FUNCTION_BLOCK AlarmNotAck (* Basic Function Block Type *)
  (* Standard: 61499-2 *)
  (* Version 0.0, 8/5/2026, Schneider Electric, Template *)
  PACKAGE SE.Nereda;
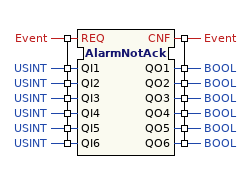
  EVENT_INPUT
    REQ WITH QI1, QI2, QI3, QI4, QI5, QI6; (* Normal Execution Request *)
  END_EVENT
  EVENT_OUTPUT
    CNF WITH QO1, QO2, QO3, QO4, QO5, QO6; (* Execution Confirmation *)
  END_EVENT
  VAR_INPUT
    QI1 : USINT; (* Input event qualifier *)
    QI2 : USINT;
    QI3 : USINT;
    QI4 : USINT;
    QI5 : USINT;
    QI6 : USINT;
  END_VAR
  VAR_OUTPUT
    QO1 : BOOL; (* Output event qualifier *)
    QO2 : BOOL;
    QO3 : BOOL;
    QO4 : BOOL;
    QO5 : BOOL;
    QO6 : BOOL;
  END_VAR
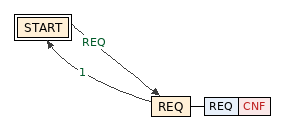
  EC_STATES
    START; (* Initial State *)
    REQ : REQ -> CNF; (* Normal execution *)
  END_STATES
  EC_TRANSITIONS
    START TO REQ := REQ;
    REQ TO START := 1;
  END_TRANSITIONS
  ALGORITHM INIT IN ST: (* Initialization algorithm *)
;
  END_ALGORITHM
  ALGORITHM REQ IN ST: (* Normally executed algorithm *)
;
IF QI1 = 2 THEN
	QO1 := TRUE;
ELSIF QI1 = 0 THEN
	QO1 := FALSE;
END_IF;

IF QI2 = 2 THEN
	QO2 := TRUE;
ELSIF QI2 = 0 THEN
	QO2 := FALSE;
END_IF;

IF QI3 = 2 THEN
	QO3 := TRUE;
ELSIF QI3 = 0 THEN
	QO3 := FALSE;
END_IF;

IF QI4 = 2 THEN
	QO4 := TRUE;
ELSIF QI4 = 0 THEN
	QO4 := FALSE;
END_IF;

IF QI5 = 2 THEN
	QO5 := TRUE;
ELSIF QI5 = 0 THEN
	QO5 := FALSE;
END_IF;

IF QI6 = 2 THEN
	QO6 := TRUE;
ELSIF QI6 = 0 THEN
	QO6 := FALSE;
END_IF;
  END_ALGORITHM
END_FUNCTION_BLOCK
